// TIA Portal project "conveyer-start-stop" (V20)

(* hardware
DEVICE "S7-1200 G2 station_1"  S7-1200 G2 Station
   slot 0: "Rack_0"  S71200G2 Rack  Rack  V1.0
   slot 1: "G2_PLC_1"  CPU 1214C DC/DC/DC  6ES7 214-1AH50-0XB0  V1.0
*)

// ===== PLC "G2_PLC_1"  CPU 1214C DC/DC/DC =====

VAR_GLOBAL   // PLC tag table "I/O"
   "Start/Stop" AT %I0.0 : Bool;
   "FaultReset" AT %I0.1 : Bool;
   "Motor" AT %Q0.0 : Bool;
   "FaultActive" AT %I0.3 : Bool;
   "EStop" AT %I0.2 : Bool;
   "FaultLatched" AT %M0.0 : Bool;
END_VAR

ORGANIZATION_BLOCK "Main"   // OB1, LAD, ProgramCycle
TITLE = "Main Program Sweep (Cycle)"
{ S7_Optimized_Access := 'TRUE' }
VERSION : 0.1
   VAR_INPUT
      Initial_Call : Bool;   // Initial call of this OB
      Remanence : Bool;   // =True, if remanent data are available
   END_VAR
BEGIN

REGION Network 1
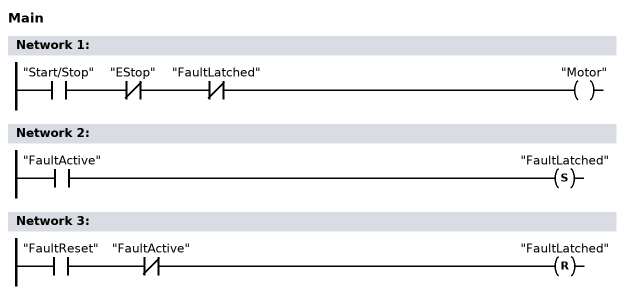
   RUNG wire#powerrail
      Contact( "Start/Stop" )
      I_Contact( "EStop" )
      I_Contact( "FaultLatched" )
      Coil( "Motor" )
   END_RUNG
   // the same network as SCL:
   "Motor" := "Start/Stop" AND NOT "EStop" AND NOT "FaultLatched";
END_REGION

REGION Network 2
   RUNG wire#powerrail
      Contact( "FaultActive" )
      S_Coil( "FaultLatched" )
   END_RUNG
   // the same network as SCL:
   IF "FaultActive" THEN "FaultLatched" := TRUE; END_IF;
END_REGION

REGION Network 3
   RUNG wire#powerrail
      Contact( "FaultReset" )
      I_Contact( "FaultActive" )
      R_Coil( "FaultLatched" )
   END_RUNG
   // the same network as SCL:
   IF "FaultReset" AND NOT "FaultActive" THEN "FaultLatched" := FALSE; END_IF;
END_REGION
END_ORGANIZATION_BLOCK